Fanuc KAREL source: kx00002.KL

-- PROVISIONAL review KL for V770-1; original PC SHA256 8e1aed2cbba2421b155da5209a7bb652907a59b183cad5db062a56ceeed9f8f0
-- Incomplete behavior may be omitted. Consult companion uncertainty JSON. Do not deploy.
PROGRAM KX00002
%NOLOCKGROUP
VAR
  I : INTEGER
  J : INTEGER
  B : BOOLEAN
  F : FILE
  S : STRING[80]
-- UNRESOLVED_DECL P type=000102
BEGIN
  -- UNRESOLVED_PC offsets 5-32; opcodes 22,3F,3F,3D
  -- UNRESOLVED_PC offsets 37-44; opcodes 22,39
  -- UNRESOLVED_PC offsets 49-53; opcodes 7F
END KX00002
